FUNCTION_BLOCK EliteBoard (* Service Interface Function Block Type *)
  (* Standard: 61499-2; Description: Copyright (c) 2021 Jonathan Lainer This program and the accompanying materials are made available under the terms of the Eclipse Public License 2.0 which is available at https://www.eclipse.org/legal/epl-2.0/ SPDX-License-Identifier: EPL-2.0 *)
  (* Version 1.0, 2021-02-22, Jonathan Lainer, Initial Contribution *)
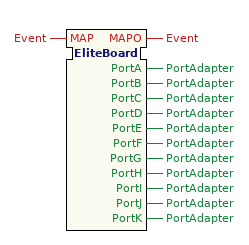
  EVENT_INPUT
    MAP;
  END_EVENT
  EVENT_OUTPUT
    MAPO;
  END_EVENT
  PLUGS
    PortA : PortAdapter;
    PortB : PortAdapter;
    PortC : PortAdapter;
    PortD : PortAdapter;
    PortE : PortAdapter;
    PortF : PortAdapter;
    PortG : PortAdapter;
    PortH : PortAdapter;
    PortI : PortAdapter;
    PortJ : PortAdapter;
    PortK : PortAdapter;
  END_PLUGS
END_FUNCTION_BLOCK
